// TIA Portal V20 export
TYPE "LER_typeCommunication"
// stored: Access Published
   STRUCT
      InspectionToStack : "LER_typeCommunicationData_I2S";
      StackToInspection : "LER_typeCommunicationData_S2I";
   END_STRUCT;
END_TYPE
